(* Logix 5000 project; controller add_ons_rslogix5000 vendor 1 type 14 code 106 rev 20.11; software revision 20.00 *)
// Repository of my personal add-ons for programming programmable logic controllers, Allen bradley.

TASK MainTask (continuous, watchdog 500 ms) : MainProgram

MODULES
   Local : vendor 1 type 14 code 106 (Compact 0, rev 20.11)
END_MODULES

TYPE Engine :
STRUCT
   START : BOOL;
   STOP : BOOL;
   RUNNING : BOOL;
   SET_SPEED : INT;
   GET_SPEED : INT;
END_STRUCT
END_TYPE

TYPE Pump :
STRUCT
   START : BOOL;
   STOP : BOOL;
   RUNNING : BOOL;
   SET_SPEED : INT;
   GET_SPEED : INT;
END_STRUCT
END_TYPE

ADD_ON_INSTRUCTION ANALOG_SCALE_IN   (* revision 1.0 *)
VAR_IN_OUT
   INPUT : INT; {required}
END_VAR
VAR_INPUT
   MAX_RESOLUTE : INT; {required}
   MIN_RESOLUTE : INT; {required}
   MAX_SCALE : INT; {required}
   MIN_SCALE : INT; {required}
END_VAR
VAR_OUTPUT
   OUTPUT_IN_ENGINEERING_UNITS : INT; {access Read Only, required}
END_VAR

ROUTINE Logic   (* ladder *)
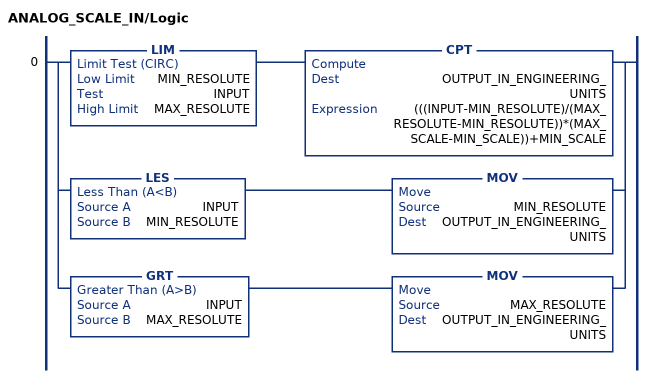
   0: [LIM(MIN_RESOLUTE,INPUT,MAX_RESOLUTE) CPT(OUTPUT_IN_ENGINEERING_UNITS,(((INPUT-MIN_RESOLUTE)/(MAX_RESOLUTE-MIN_RESOLUTE))*(MAX_SCALE-MIN_SCALE))+MIN_SCALE) ,LES(INPUT,MIN_RESOLUTE) MOV(MIN_RESOLUTE,OUTPUT_IN_ENGINEERING_UNITS) ,GRT(INPUT,MAX_RESOLUTE) MOV(MAX_RESOLUTE,OUTPUT_IN_ENGINEERING_UNITS) ];
END_ROUTINE
END_ADD_ON_INSTRUCTION

ADD_ON_INSTRUCTION ANALOG_SCALE_OUT   (* revision 1.0, vendor Daniel A. Villena H. *)
VAR_INPUT
   INPUT_IN_ENGINEERING_UNITS : INT; {required}
   MAX_RESOLUTE : INT; {required}
   MIN_RESOLUTE : INT; {required}
   MAX_SCALE : INT; {required}
   MIN_SCALE : INT; {required}
END_VAR
VAR_IN_OUT
   OUTPUT : INT; {required}
END_VAR

ROUTINE Logic   (* ladder *)
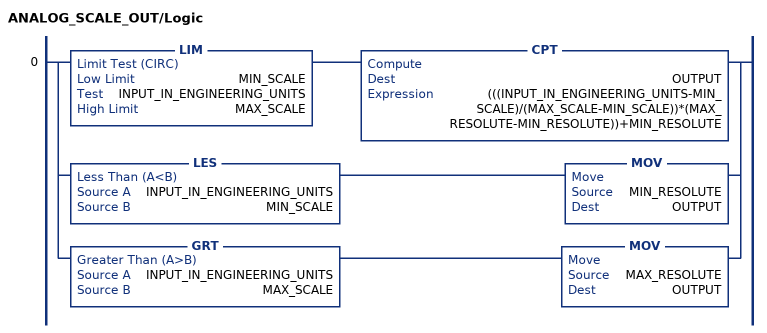
   0: [LIM(MIN_SCALE,INPUT_IN_ENGINEERING_UNITS,MAX_SCALE) CPT(OUTPUT,(((INPUT_IN_ENGINEERING_UNITS-MIN_SCALE)/(MAX_SCALE-MIN_SCALE))*(MAX_RESOLUTE-MIN_RESOLUTE))+MIN_RESOLUTE) ,LES(INPUT_IN_ENGINEERING_UNITS,MIN_SCALE) MOV(MIN_RESOLUTE,OUTPUT) ,GRT(INPUT_IN_ENGINEERING_UNITS,MAX_SCALE) MOV(MAX_RESOLUTE,OUTPUT) ];
END_ROUTINE
END_ADD_ON_INSTRUCTION

ADD_ON_INSTRUCTION HOA_Control   (* revision 1.0, vendor Daniel A. Villena H. *)
// Management of the operating system.
// 0 = OFF
// 1 = HAND
// 2 = AUTO
// Revision note:
// Initial Version
VAR_IN_OUT
   HAND : BOOL; {required}
   OFF : BOOL; {required}
   AUTO : BOOL; {required}
END_VAR
VAR_OUTPUT
   CONTROL : SINT; {access Read Only, required}
END_VAR
VAR
   ONS0 : BOOL; {access None}
   ONS1 : BOOL; {access None}
   ONS2 : BOOL; {access None}
END_VAR

ROUTINE Logic   (* ladder *)
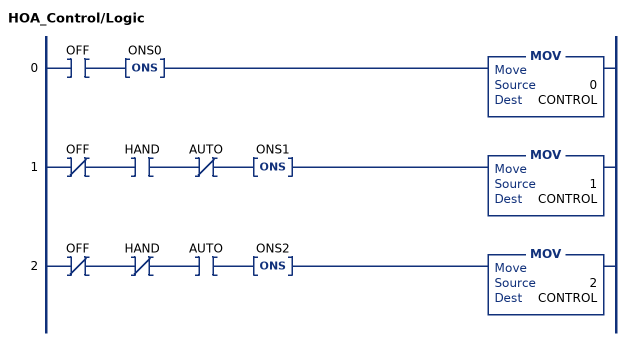
   0: XIC(OFF)ONS(ONS0)MOV(0,CONTROL);
   1: XIO(OFF)XIC(HAND)XIO(AUTO)ONS(ONS1)MOV(1,CONTROL);
   2: XIO(OFF)XIO(HAND)XIC(AUTO)ONS(ONS2)MOV(2,CONTROL);
END_ROUTINE
END_ADD_ON_INSTRUCTION

ADD_ON_INSTRUCTION OOF_Control   (* revision 1.0, vendor Daniel A. Villena H. *)
// Management of the operating system.
// 0 = FAULTED
// 1 = RUNNING
// Revision note:
// Initial Version
VAR_INPUT
   HOA : SINT; {required}   // 0 = OFF 1 = HAND 2 = AUTO
   ALARM : BOOL; {required}
END_VAR
VAR_OUTPUT
   CONTROL : BOOL; {required}   // 0 = FAULTED 1 = RUNNING
END_VAR
VAR
   ONS1 : BOOL; {access None}
   ERROR : BOOL; {access None}
END_VAR

ROUTINE Logic   (* ladder *)
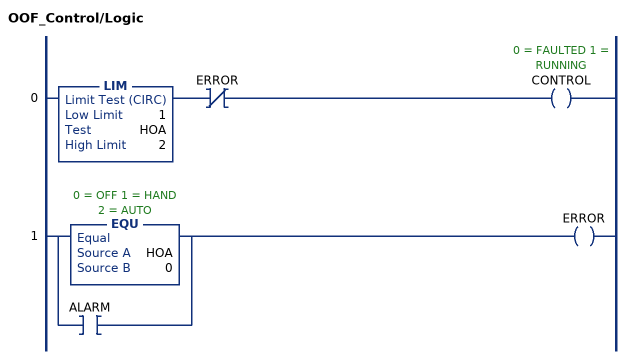
   0: LIM(1,HOA,2)XIO(ERROR)OTE(CONTROL);
   1: [EQU(HOA,0) ,XIC(ALARM) ]OTE(ERROR);
END_ROUTINE
END_ADD_ON_INSTRUCTION

PROGRAM MainProgram   (* main routine MainRoutine *)

ROUTINE MainRoutine   (* ladder *)
END_ROUTINE
END_PROGRAM
